FUNCTION_BLOCK myCompositeBlock (* Composite FB wrapping other FBs *)
  (* Standard: 61499-2 *)
  (* Version 1.0, 2025-07-11, dakudryashev *)
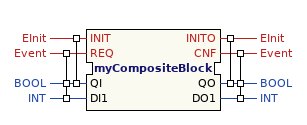
  EVENT_INPUT
    INIT : EInit WITH QI; (* Initialization Request *)
    REQ WITH QI, DI1; (* Normal Execution Request *)
  END_EVENT
  EVENT_OUTPUT
    INITO : EInit WITH QO; (* Initialization Confirm *)
    CNF WITH QO, DO1; (* Execution Confirmation *)
  END_EVENT
  VAR_INPUT
    QI : BOOL; (* Input event qualifier *)
    DI1 : INT;
  END_VAR
  VAR_OUTPUT
    QO : BOOL; (* Output event qualifier *)
    DO1 : INT;
  END_VAR
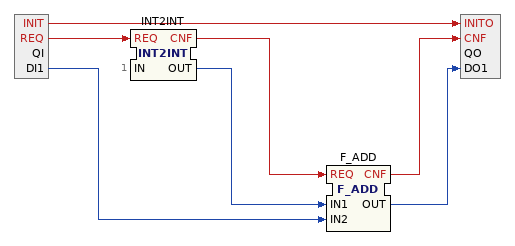
  FBS
    INT2INT : INT2INT(IN := 1);
    F_ADD : F_ADD;
  END_FBS
  EVENT_CONNECTIONS
    REQ TO INT2INT.REQ;
    INT2INT.CNF TO F_ADD.REQ;
    F_ADD.CNF TO CNF;
    INIT TO INITO;
  END_CONNECTIONS
  DATA_CONNECTIONS
    INT2INT.OUT TO F_ADD.IN1;
    DI1 TO F_ADD.IN2;
    F_ADD.OUT TO DO1;
  END_CONNECTIONS
END_FUNCTION_BLOCK
